Staubli VAL3: OnF6.pgx

program OnF6()
  local string l_sProperty[2]
  local string l_sItem
begin
  switch nPage
    case 0
      l_sProperty[0]="设置"
      l_sProperty[1]="取消"
      call user:SetProerty("",26,9,6,2,l_sProperty,l_sItem)
      if l_sItem==l_sProperty[0]
        if sItem==""
          popUpMsg("没有产品")
        else
          PublicData:sStartPrd=sItem
          PublicData:libSave()
          popUpMsg("选择产品"+sItem+"为自启动")

        endIf
      else
        PublicData:sStartPrd=""
        PublicData:libSave()
        popUpMsg("自启动取消")
      endIf
      bUserRefresh=bListRefresh=true
    break
    case 1
    break
  endSwitch
end
